Staubli VAL3: Record1.pgx

public program Record1(tool x_tTool, pointRx x_pPoint, num x_nDia)
  local string l_sString
  local num l_ni
  local num l_nVel
  local point l_pPoint[3]
  local num l_nNum[3]
begin
  //
  wait(bRecord==true and !isEmpty())
  l_ni=1
  l_sString=""
  do
    l_pPoint[0]=here(x_tTool,world)
    //cmd 与半径差值
    l_nNum[0]=distance(l_pPoint[0],x_pPoint)-x_nDia/2
    //fbk与半径差值
    l_pPoint[1]=$getPosFbk(x_tTool,world)
    l_nNum[1]=distance(l_pPoint[1],x_pPoint)-x_nDia/2
    //cmd 与 fbk
    l_nNum[2]=distance(l_pPoint[0],l_pPoint[1])
    l_sString=toString(".5",l_nNum[0])+","+toString(".5",l_nNum[1])+","+toString(".5",l_nNum[2])
    call WriteFile(l_sString)
    delay(0)
  until isEmpty()==true
  bRecord=false
end
